Yaskawa INFORM job: R1_W01(KAMERA)(0,-90)NEW.JBI

/JOB
//NAME R1_W01(KAMERA)(0,-90)NEW
///FOLDERNAME SCIANA-NOWY-R2-KM
//POS
///NPOS 9,9,0,0,0,0
///TOOL 0
///POSTYPE PULSE
///LIMIT ON
///PULSE
C00000=3259,-159822,-135039,-10688,361,-77457
///LIMIT OFF
C00001=3259,-159822,-135039,-10688,361,-77457
C00002=118675,-45665,-102005,-21757,75350,-73909
C00003=180273,41623,-63008,-27819,115689,-72022
C00004=168830,48116,-33495,-18105,111077,-70088
C00005=164695,62063,-17563,-16410,107934,-70731
C00006=169685,37723,-34985,-25566,92727,-69804
C00007=177047,21649,-54490,-29233,98284,-69028
C00008=169262,14064,-103081,-21827,78231,-74428
BC00000=161517,768606,1042197
BC00001=161517,1190244,1042197
BC00002=284380,1205478,1059252
BC00003=349545,1213558,1068298
BC00004=343588,1213558,1068298
BC00005=343588,1213558,1068298
BC00006=343588,1213558,1068298
BC00007=343753,1213558,1068298
BC00008=383547,1212278,1068298
//INST
///DATE 2024/07/16 20:05
///ATTR SC,RW
///GROUP1 RB1,BS1
NOP
'r1_W01(kamera)(0,-90)
'Path W401
SFTOF
MOVJ C00000 BC00000 VJ=100.00
MOVJ C00001 BC00001 VJ=100.00
MOVJ C00002 BC00002 VJ=100.00
MOVJ C00003 BC00003 VJ=70.00
MOVJ C00004 BC00004 VJ=20.00
MACRO1 MJ#(0) ARGF6
ARCON
MOVL C00005 BC00005 V=10.0
MOVL C00006 BC00006 V=10.0
ARCOF
MOVL C00007 BC00007 V=333.3
MOVJ C00008 BC00008 VJ=100.00
END
